{attribute 'qualified_only'}
VAR_GLOBAL
    Event_OnError : TEvent_ExecutionFailed;
    Event_OnAbort : TEvent_ExecutionAborted;
END_VAR

(* stored: Version 1.1.0.1, ProductVersion 3.1.4024.3
   GVL Events: Id {64546398-db5d-0d66-2782-a6500d59e54d} *)
